# EPICS substitutions: db/generated/scifi_bias.substitutions
# AUTO-GENERATED FILE - DO NOT EDIT
# Generated by scripts/generate_scifi_bias_substitutions.py
# Source: data/scifi_bias.csv
# Physical SiPM channels: 224
#
# P, OFF_THRESHOLD, BIAS_TOLERANCE and INITIAL_BIAS
# are supplied by dbLoadTemplate() in st.cmd.

file "db/scifi_bias.template"
{
    pattern
    {
        CHAMBER,ID,SFP,DEV
    }

    { FHF1,1,0,0 }
    { FHF1,1,0,1 }
    { FHF1,1,0,2 }
    { FHF1,1,0,3 }
    { FHF1,1,0,4 }
    { FHF1,1,0,5 }
    { FHF1,1,1,0 }
    { FHF1,1,1,1 }
    { FHF1,1,2,0 }
    { FHF1,1,2,1 }
    { FHF1,1,2,2 }
    { FHF1,1,2,3 }
    { FHF1,1,2,4 }
    { FHF1,1,2,5 }
    { FHF1,1,3,0 }
    { FHF1,1,3,1 }
    { FHF1,2,0,0 }
    { FHF1,2,0,1 }
    { FHF1,2,0,2 }
    { FHF1,2,0,3 }
    { FHF1,2,0,4 }
    { FHF1,2,0,5 }
    { FHF1,2,1,0 }
    { FHF1,2,1,1 }
    { FHF1,2,2,0 }
    { FHF1,2,2,1 }
    { FHF1,2,2,2 }
    { FHF1,2,2,3 }
    { FHF1,2,2,4 }
    { FHF1,2,2,5 }
    { FHF1,2,3,0 }
    { FHF1,2,3,1 }
    { FHF1,3,0,0 }
    { FHF1,3,0,1 }
    { FHF1,3,0,2 }
    { FHF1,3,0,3 }
    { FHF1,3,0,4 }
    { FHF1,3,0,5 }
    { FHF1,3,1,0 }
    { FHF1,3,1,1 }
    { FHF1,3,2,0 }
    { FHF1,3,2,1 }
    { FHF1,3,2,2 }
    { FHF1,3,2,3 }
    { FHF1,3,2,4 }
    { FHF1,3,2,5 }
    { FHF1,3,3,0 }
    { FHF1,3,3,1 }
    { FMF1,1,0,0 }
    { FMF1,1,0,1 }
    { FMF1,1,0,2 }
    { FMF1,1,0,3 }
    { FMF1,1,0,4 }
    { FMF1,1,0,5 }
    { FMF1,1,1,0 }
    { FMF1,1,1,1 }
    { FMF1,1,2,0 }
    { FMF1,1,2,1 }
    { FMF1,1,2,2 }
    { FMF1,1,2,3 }
    { FMF1,1,2,4 }
    { FMF1,1,2,5 }
    { FMF1,1,3,0 }
    { FMF1,1,3,1 }
    { FMF1,2,0,0 }
    { FMF1,2,0,1 }
    { FMF1,2,0,2 }
    { FMF1,2,0,3 }
    { FMF1,2,0,4 }
    { FMF1,2,0,5 }
    { FMF1,2,1,0 }
    { FMF1,2,1,1 }
    { FMF1,2,2,0 }
    { FMF1,2,2,1 }
    { FMF1,2,2,2 }
    { FMF1,2,2,3 }
    { FMF1,2,2,4 }
    { FMF1,2,2,5 }
    { FMF1,2,3,0 }
    { FMF1,2,3,1 }
    { FMF2,1,0,0 }
    { FMF2,1,0,1 }
    { FMF2,1,0,2 }
    { FMF2,1,0,3 }
    { FMF2,1,0,4 }
    { FMF2,1,0,5 }
    { FMF2,1,1,0 }
    { FMF2,1,1,1 }
    { FMF2,1,2,0 }
    { FMF2,1,2,1 }
    { FMF2,1,2,2 }
    { FMF2,1,2,3 }
    { FMF2,1,2,4 }
    { FMF2,1,2,5 }
    { FMF2,1,3,0 }
    { FMF2,1,3,1 }
    { FMF2,2,0,0 }
    { FMF2,2,0,1 }
    { FMF2,2,0,2 }
    { FMF2,2,0,3 }
    { FMF2,2,0,4 }
    { FMF2,2,0,5 }
    { FMF2,2,1,0 }
    { FMF2,2,1,1 }
    { FMF2,2,2,0 }
    { FMF2,2,2,1 }
    { FMF2,2,2,2 }
    { FMF2,2,2,3 }
    { FMF2,2,2,4 }
    { FMF2,2,2,5 }
    { FMF2,2,3,0 }
    { FMF2,2,3,1 }
    { FMF3,1,0,0 }
    { FMF3,1,0,1 }
    { FMF3,1,0,2 }
    { FMF3,1,0,3 }
    { FMF3,1,0,4 }
    { FMF3,1,0,5 }
    { FMF3,1,1,0 }
    { FMF3,1,1,1 }
    { FMF3,1,2,0 }
    { FMF3,1,2,1 }
    { FMF3,1,2,2 }
    { FMF3,1,2,3 }
    { FMF3,1,2,4 }
    { FMF3,1,2,5 }
    { FMF3,1,3,0 }
    { FMF3,1,3,1 }
    { FMF3,2,0,0 }
    { FMF3,2,0,1 }
    { FMF3,2,0,2 }
    { FMF3,2,0,3 }
    { FMF3,2,0,4 }
    { FMF3,2,0,5 }
    { FMF3,2,1,0 }
    { FMF3,2,1,1 }
    { FMF3,2,2,0 }
    { FMF3,2,2,1 }
    { FMF3,2,2,2 }
    { FMF3,2,2,3 }
    { FMF3,2,2,4 }
    { FMF3,2,2,5 }
    { FMF3,2,3,0 }
    { FMF3,2,3,1 }
    { FPF2,1,0,0 }
    { FPF2,1,0,1 }
    { FPF2,1,0,2 }
    { FPF2,1,0,3 }
    { FPF2,1,0,4 }
    { FPF2,1,0,5 }
    { FPF2,1,1,0 }
    { FPF2,1,1,1 }
    { FPF2,1,2,0 }
    { FPF2,1,2,1 }
    { FPF2,1,2,2 }
    { FPF2,1,2,3 }
    { FPF2,1,2,4 }
    { FPF2,1,2,5 }
    { FPF2,1,3,0 }
    { FPF2,1,3,1 }
    { FPF2,2,0,0 }
    { FPF2,2,0,1 }
    { FPF2,2,0,2 }
    { FPF2,2,0,3 }
    { FPF2,2,0,4 }
    { FPF2,2,0,5 }
    { FPF2,2,1,0 }
    { FPF2,2,1,1 }
    { FPF2,2,2,0 }
    { FPF2,2,2,1 }
    { FPF2,2,2,2 }
    { FPF2,2,2,3 }
    { FPF2,2,2,4 }
    { FPF2,2,2,5 }
    { FPF2,2,3,0 }
    { FPF2,2,3,1 }
    { FPF3,1,0,0 }
    { FPF3,1,0,1 }
    { FPF3,1,0,2 }
    { FPF3,1,0,3 }
    { FPF3,1,0,4 }
    { FPF3,1,0,5 }
    { FPF3,1,1,0 }
    { FPF3,1,1,1 }
    { FPF3,1,2,0 }
    { FPF3,1,2,1 }
    { FPF3,1,2,2 }
    { FPF3,1,2,3 }
    { FPF3,1,2,4 }
    { FPF3,1,2,5 }
    { FPF3,1,3,0 }
    { FPF3,1,3,1 }
    { FPF4,1,0,0 }
    { FPF4,1,0,1 }
    { FPF4,1,0,2 }
    { FPF4,1,0,3 }
    { FPF4,1,0,4 }
    { FPF4,1,0,5 }
    { FPF4,1,1,0 }
    { FPF4,1,1,1 }
    { FPF4,1,2,0 }
    { FPF4,1,2,1 }
    { FPF4,1,2,2 }
    { FPF4,1,2,3 }
    { FPF4,1,2,4 }
    { FPF4,1,2,5 }
    { FPF4,1,3,0 }
    { FPF4,1,3,1 }
    { FPF4,2,0,0 }
    { FPF4,2,0,1 }
    { FPF4,2,0,2 }
    { FPF4,2,0,3 }
    { FPF4,2,0,4 }
    { FPF4,2,0,5 }
    { FPF4,2,1,0 }
    { FPF4,2,1,1 }
    { FPF4,2,2,0 }
    { FPF4,2,2,1 }
    { FPF4,2,2,2 }
    { FPF4,2,2,3 }
    { FPF4,2,2,4 }
    { FPF4,2,2,5 }
    { FPF4,2,3,0 }
    { FPF4,2,3,1 }
}
